// TIA Portal V17 export
// export: Created 2022-12-09T10:51:18.3245614Z, ExportSetting WithDefaults, DisplayName Totally Integrated Automation Portal, DisplayVersion V17 Update 5, DisplayName TIA Portal Openness, DisplayVersion V17 Update 5, DisplayName TIA Portal Version Control Interface, DisplayVersion V17, DisplayName Simotion SCOUT TIA, DisplayVersion 5.4.3.0, DisplayName SINAMICS Startdrive Advanced, DisplayVersion V17 SP1, DisplayName SINAMICS Startdrive G130, G150, S120, S150, SINAMICS MV, S210, DisplayVersion V17 SP1, DisplayName SINAMICS Startdrive G110M, G120, G120C, G120D, G120P, G115D, DisplayVersion V17 SP1, DisplayName STEP 7 Professional, DisplayVersion V17 Update 5, DisplayName STEP 7 Safety, DisplayVersion V17, DisplayName WinCC Advanced, DisplayVersion V17 Update 5
TYPE "UDT_UserManagement"
// stored: IsFailsafeCompliant false
   STRUCT
      Valid : Bool;
      UserName : String;
      Password : String;
      "LogOff-Time" : DInt := 10;
      AuthorisationGroup : Int;
      Authorisation : "UDT_UserAuthorisation";
   END_STRUCT;
END_TYPE
